Omron CX-Programmer project NewProject (CX-Programmer 9.81)

# PLC Exercicio_Movimento_da_carrinha: CP1L-E EM

## Program NewProgram1 (cyclic task 0)
Local symbols
AV 100.04 BOOL  ; Abrir valvula
Etapa_0 2.00 BOOL  ; Etapa 0 do Grafcet
Etapa_1 2.01 BOOL  ; Etapa 1 do Grafcet
Etapa_2 2.02 BOOL  ; Etapa 2 do Grafcet
Etapa_3 2.03 BOOL  ; Etapa 3 do Grafcet
Etapa_4 2.04 BOOL  ; Etapa 4 do Grafcet
Etapa_5 2.05 BOOL  ; Etapa 5 do Grafcet
FV 100.05 BOOL  ; Fechar valvula
Flag_T T0001 BOOL  ; Flag do Temporizador
Motor_D 100.02 BOOL  ; Motor move para direita
Motor_E 100.03 BOOL  ; Motor move para esquerda
Motor_L 100.00 BOOL  ; Ligar motor
Motor_P 100.01 BOOL  ; Parar motor
Peso 0.04 BOOL  ; Sensor de peso
Sa 0.03 BOOL  ; Sensor fim de curso esquerdo
Sb 0.02 BOOL  ; Sensor fim de curso direito
Start 0.00 BOOL  ; Botao Start
Stop 0.01 BOOL  ; Botao Stop
T 1 NUMBER  ; Temporizador
Tempo_T #50 NUMBER  ; Tempo do Temporizador - 5 segundos

### Section Main

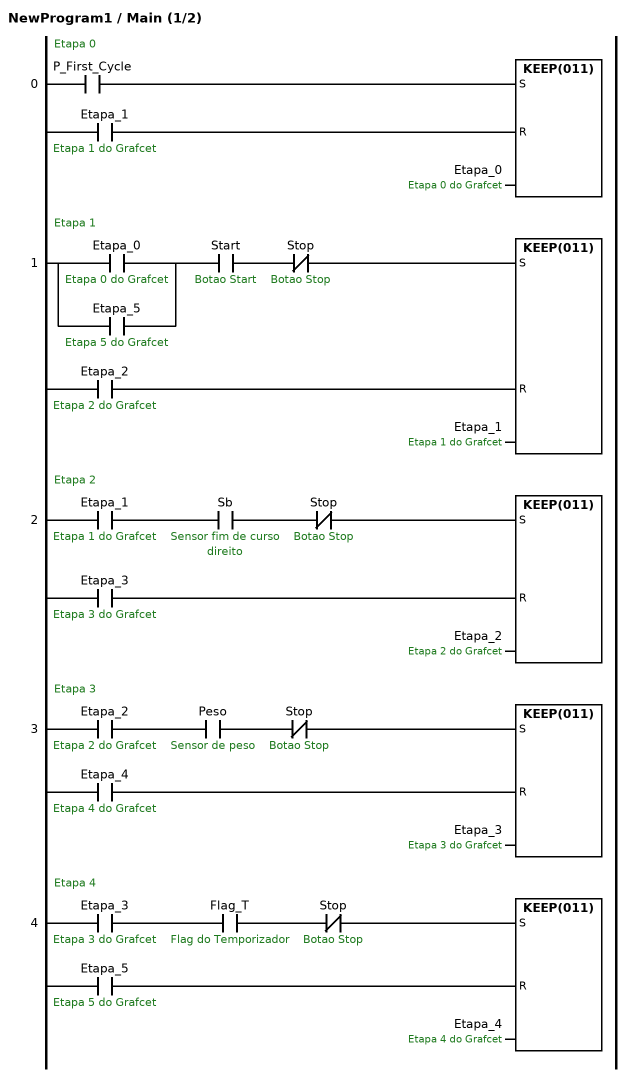
; rung 0: Etapa 0
LD P_First_Cycle
LD Etapa_1  ; Etapa 1 do Grafcet
KEEP(011) Etapa_0  ; Etapa 0 do Grafcet
; rung 1: Etapa 1
LD Etapa_0  ; Etapa 0 do Grafcet
OR Etapa_5  ; Etapa 5 do Grafcet
AND Start  ; Botao Start
ANDNOT Stop  ; Botao Stop
LD Etapa_2  ; Etapa 2 do Grafcet
KEEP(011) Etapa_1  ; Etapa 1 do Grafcet
; rung 2: Etapa 2
LD Etapa_1  ; Etapa 1 do Grafcet
AND Sb  ; Sensor fim de curso direito
ANDNOT Stop  ; Botao Stop
LD Etapa_3  ; Etapa 3 do Grafcet
KEEP(011) Etapa_2  ; Etapa 2 do Grafcet
; rung 3: Etapa 3
LD Etapa_2  ; Etapa 2 do Grafcet
AND Peso  ; Sensor de peso
ANDNOT Stop  ; Botao Stop
LD Etapa_4  ; Etapa 4 do Grafcet
KEEP(011) Etapa_3  ; Etapa 3 do Grafcet
; rung 4: Etapa 4
LD Etapa_3  ; Etapa 3 do Grafcet
AND Flag_T  ; Flag do Temporizador
ANDNOT Stop  ; Botao Stop
LD Etapa_5  ; Etapa 5 do Grafcet
KEEP(011) Etapa_4  ; Etapa 4 do Grafcet

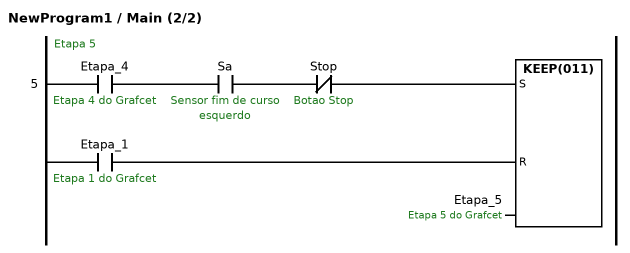
; rung 5: Etapa 5
LD Etapa_4  ; Etapa 4 do Grafcet
AND Sa  ; Sensor fim de curso esquerdo
ANDNOT Stop  ; Botao Stop
LD Etapa_1  ; Etapa 1 do Grafcet
KEEP(011) Etapa_5  ; Etapa 5 do Grafcet

### Section Out

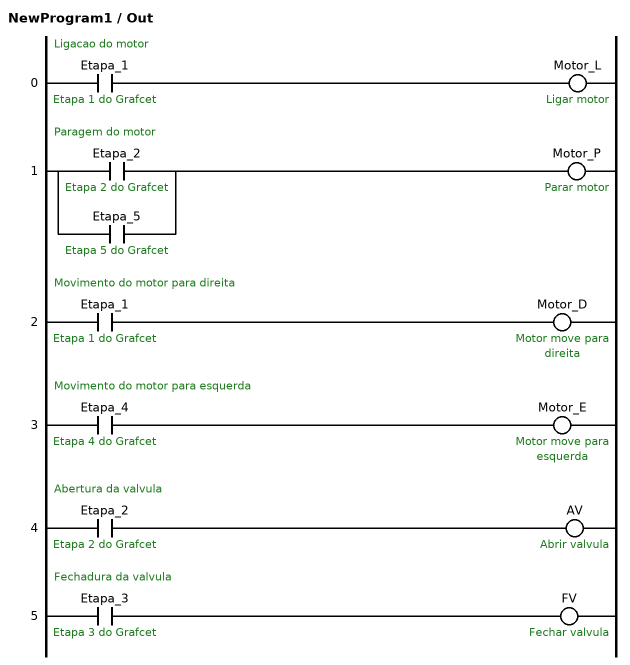
; rung 0: Ligacao do motor
LD Etapa_1  ; Etapa 1 do Grafcet
OUT Motor_L  ; Ligar motor
; rung 1: Paragem do motor
LD Etapa_2  ; Etapa 2 do Grafcet
OR Etapa_5  ; Etapa 5 do Grafcet
OUT Motor_P  ; Parar motor
; rung 2: Movimento do motor para direita
LD Etapa_1  ; Etapa 1 do Grafcet
OUT Motor_D  ; Motor move para direita
; rung 3: Movimento do motor para esquerda
LD Etapa_4  ; Etapa 4 do Grafcet
OUT Motor_E  ; Motor move para esquerda
; rung 4: Abertura da valvula
LD Etapa_2  ; Etapa 2 do Grafcet
OUT AV  ; Abrir valvula
; rung 5: Fechadura da valvula
LD Etapa_3  ; Etapa 3 do Grafcet
OUT FV  ; Fechar valvula

### Section Timer

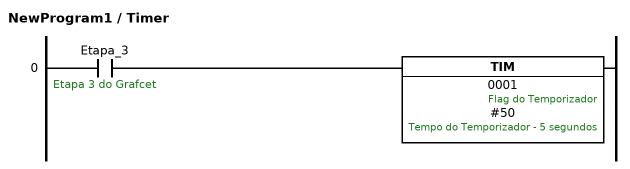
; rung 0
LD Etapa_3  ; Etapa 3 do Grafcet
TIM 0001 #50  ; Tempo do Temporizador - 5 segundos, Flag do Temporizador

### Section END
; rung 0
END(001)